// TIA Portal V15.1 export
// export: Created 2024-05-17T05:38:33.7575808Z, ExportSetting WithDefaults, DisplayName Totally Integrated Automation Portal, DisplayVersion V15.1 Update 5, DisplayName TIA Portal Openness, DisplayVersion V15.1 Update 5, DisplayName SINAMICS Startdrive Advanced, DisplayVersion V15.1, DisplayName G130, G150, S120, S150, SINAMICS MV, S210, DisplayVersion V15.1, DisplayName G110M, G120, G120C, G120D, G120P, DisplayVersion V15.1, DisplayName STEP 7 Professional, DisplayVersion V15.1 Update 5, DisplayName STEP 7 Safety, DisplayVersion V15.1, DisplayName WinCC Professional, DisplayVersion V15.1 Update 5, DisplayName SIMATIC Visualization Architect, DisplayVersion V15.1
FUNCTION_BLOCK "LProcMonStabValv"   // FB1701, FBD
TITLE = LProcMonStabValv
{ S7_Optimized_Access := 'FALSE' }
AUTHOR : VCC
FAMILY : ProcEqp
NAME : ProcValv
VERSION : 1.0
// ================================================================================
// This module is used to activate a monostable valve. It includes its own Mode 
// function. There is the possibility to use it normally open or normally closed, 
// with or without closed and open detections.
// ================================================================================
// stored: AutoNumber false, IsIECCheckEnabled false, SetENOAutomatically False, UDAEnableTagReadback false
   VAR_INPUT
      I_MaxTime { ExternalAccessible := 'False'; ExternalVisible := 'False'; ExternalWritable := 'False'} : DInt;   // Maximum Time to get Set and reset detections
      I_DetSet { ExternalAccessible := 'False'; ExternalVisible := 'False'; ExternalWritable := 'False'} : Bool;   // Detection SET
      I_DetReset { ExternalAccessible := 'False'; ExternalVisible := 'False'; ExternalWritable := 'False'} : Bool;   // Detection RESET
      I_EnableAlarm { ExternalAccessible := 'False'; ExternalVisible := 'False'; ExternalWritable := 'False'} : Bool;   // Enable Alarm for the Acof detections
      I_AutoReq { ExternalAccessible := 'False'; ExternalVisible := 'False'; ExternalWritable := 'False'} : Bool;   // Auto Request from equation or Sequence
      I_InterlockOk { ExternalAccessible := 'False'; ExternalVisible := 'False'; ExternalWritable := 'False'} : Bool;   // Interlock
      I_PBSetPBResetAllAutoSel { ExternalAccessible := 'False'; ExternalVisible := 'False'; ExternalWritable := 'False'} : Struct   // Set PB activated - Reset PB activated - All HMI Auto selected
         HMI1SetPB { ExternalAccessible := 'False'; ExternalVisible := 'False'; ExternalWritable := 'False'} : Bool;   // Set PB activated on HMI1
         HMI1ResetPB { ExternalAccessible := 'False'; ExternalVisible := 'False'; ExternalWritable := 'False'} : Bool;   // Reset PB activated on HMI1
         HMI1AllHMIAutoSel { ExternalAccessible := 'False'; ExternalVisible := 'False'; ExternalWritable := 'False'} : Bool;   // All HMI Auto selected on HMI1
         HMI2SetPB { ExternalAccessible := 'False'; ExternalVisible := 'False'; ExternalWritable := 'False'} : Bool;   // Set PB activated on HMI2
         HMI2ResetPB { ExternalAccessible := 'False'; ExternalVisible := 'False'; ExternalWritable := 'False'} : Bool;   // Reset PB activated on HMI2
         HMI2AllHMIAutoSel { ExternalAccessible := 'False'; ExternalVisible := 'False'; ExternalWritable := 'False'} : Bool;   // All HMI Auto selected on HMI2
         HMI3SetPB { ExternalAccessible := 'False'; ExternalVisible := 'False'; ExternalWritable := 'False'} : Bool;   // Set PB activated on HMI3
         HMI3ResetPB { ExternalAccessible := 'False'; ExternalVisible := 'False'; ExternalWritable := 'False'} : Bool;   // Reset PB activated on HMI3
         HMI3AllHMIAutoSel { ExternalAccessible := 'False'; ExternalVisible := 'False'; ExternalWritable := 'False'} : Bool;   // All HMI Auto selected on HMI3
         HMI4SetPB { ExternalAccessible := 'False'; ExternalVisible := 'False'; ExternalWritable := 'False'} : Bool;   // Set PB activated on HMI4
         HMI4ResetPB { ExternalAccessible := 'False'; ExternalVisible := 'False'; ExternalWritable := 'False'} : Bool;   // Reset PB activated on HMI4
         HMI4AllHMIAutoSel { ExternalAccessible := 'False'; ExternalVisible := 'False'; ExternalWritable := 'False'} : Bool;   // All HMI Auto selected on HMI4
         HMI5SetPB { ExternalAccessible := 'False'; ExternalVisible := 'False'; ExternalWritable := 'False'} : Bool;   // Set PB activated on HMI5
         HMI5ResetPB { ExternalAccessible := 'False'; ExternalVisible := 'False'; ExternalWritable := 'False'} : Bool;   // Reset PB activated on HMI5
         HMI5AllHMIAutoSel { ExternalAccessible := 'False'; ExternalVisible := 'False'; ExternalWritable := 'False'} : Bool;   // All HMI Auto selected on HMI5
         StartPBSel { ExternalAccessible := 'False'; ExternalVisible := 'False'; ExternalWritable := 'False'} : Bool;   // Start is activated
         AlarmResetPBSel { ExternalAccessible := 'False'; ExternalVisible := 'False'; ExternalWritable := 'False'} : Bool;   // Alarm reset is activated
      END_STRUCT;
      I_UpperLevelAlarmA { ExternalAccessible := 'False'; ExternalVisible := 'False'; ExternalWritable := 'False'} : Bool;   // Alarm A active from the top level
      I_UpperLevelAlarmB { ExternalAccessible := 'False'; ExternalVisible := 'False'; ExternalWritable := 'False'} : Bool;   // Alarm B active from the top level
      C_EnableSetResetHMI { ExternalAccessible := 'False'; ExternalVisible := 'False'; ExternalWritable := 'False'} : Bool;   // Enable Set-Reset functions from HMI
      C_ManualForcedUsed { ExternalAccessible := 'False'; ExternalVisible := 'False'; ExternalWritable := 'False'} : Bool;   // Manual Forced is used (=true)
      C_SelfHolding { ExternalAccessible := 'False'; ExternalVisible := 'False'; ExternalWritable := 'False'} : Bool := TRUE;   // Enable SelfHolding Command
      C_DetSetUsed { ExternalAccessible := 'False'; ExternalVisible := 'False'; ExternalWritable := 'False'} : Bool;   // Detection SET used (true=used)
      C_DetResetUsed { ExternalAccessible := 'False'; ExternalVisible := 'False'; ExternalWritable := 'False'} : Bool;   // Detection RESET used (true=used)
      C_ValveNO { ExternalAccessible := 'False'; ExternalVisible := 'False'; ExternalWritable := 'False'} : Bool;   // Valve Normally Open (NO=true)
   END_VAR
   VAR_OUTPUT
      O_ValveCmd { ExternalAccessible := 'False'; ExternalVisible := 'False'; ExternalWritable := 'False'} : Bool;   // Valve Command
      O_AlarmABCondition { ExternalAccessible := 'False'; ExternalVisible := 'False'; ExternalWritable := 'False'} : Bool;   // Alarm AB condition
      O_AlarmA { ExternalAccessible := 'False'; ExternalVisible := 'False'; ExternalWritable := 'False'} : Bool;   // Summary Alarm A from the Valve
      O_AlarmB { ExternalAccessible := 'False'; ExternalVisible := 'False'; ExternalWritable := 'False'} : Bool;   // Summary Alarm B from the Valve
      O_AlarmC { ExternalAccessible := 'False'; ExternalVisible := 'False'; ExternalWritable := 'False'} : Bool;   // Summary Alarm C from the Valve
      O_AlarmD { ExternalAccessible := 'False'; ExternalVisible := 'False'; ExternalWritable := 'False'} : Bool;   // Summary Alarm D from the Valve
      H_IAnim { ExternalAccessible := 'False'; ExternalVisible := 'False'; ExternalWritable := 'False'} : Word;   // HMI Animation of the icon
      H_AlarmWord { ExternalAccessible := 'False'; ExternalVisible := 'False'; ExternalWritable := 'False'} : DWord;   // Alarm Word
   END_VAR
   VAR DB_SPECIFIC
      AB_OverTimeAutoSel { ExternalAccessible := 'False'; ExternalVisible := 'False'; ExternalWritable := 'False'} : Bool;   // Alarm Overtime Auto selected
      AB_AcofDetSet { ExternalAccessible := 'False'; ExternalVisible := 'False'; ExternalWritable := 'False'} : Bool;   // Acof Fault Set detection
      AB_AcofDetReset { ExternalAccessible := 'False'; ExternalVisible := 'False'; ExternalWritable := 'False'} : Bool;   // Acof Fault Reset detection
      AD_InterlockAlarm { ExternalAccessible := 'False'; ExternalVisible := 'False'; ExternalWritable := 'False'} : Bool;   // Interlock Fault
      H_HMIModeCmd : Word;   // Mode commands from HMI
      H_ActiveHMI : Int;   // Active HMI
      H_NameActiveHMI : String[25];   // Name of the Active HMI
      H_Out : Struct   // HMI
         DetSetIAnim : Word;   // HMI Animation of the Detection
         DetResetIAnim : Word;   // HMI Animation of the Detection
         OutputIAnim : Word;   // HMI Animation of the output
         Anim : Word;   // HMI Animation of the object
         Anim2 : Word;   // HMI Animation of the object
         Anim3 : Bool;   // HMI Animation bool
         DBnr : Int;   // HMI Animation DB number
      END_STRUCT;
      OverTimeAutoSelCond { ExternalAccessible := 'False'; ExternalVisible := 'False'; ExternalWritable := 'False'} : Bool;   // Overtime Auto selected condition
      AcofDetSetCond { ExternalAccessible := 'False'; ExternalVisible := 'False'; ExternalWritable := 'False'} : Bool;   // Acof Detection set condition
      AcofDetResetCond { ExternalAccessible := 'False'; ExternalVisible := 'False'; ExternalWritable := 'False'} : Bool;   // Acof Detection reset condition
      AutoMode { ExternalAccessible := 'False'; ExternalVisible := 'False'; ExternalWritable := 'False'} : Bool;   // Auto mode
      ManualMode { ExternalAccessible := 'False'; ExternalVisible := 'False'; ExternalWritable := 'False'} : Bool;   // Manual mode
      AutoModeSel { ExternalAccessible := 'False'; ExternalVisible := 'False'; ExternalWritable := 'False'} : Bool;   // Auto Mode Selection from HMI
      ManualModeSel { ExternalAccessible := 'False'; ExternalVisible := 'False'; ExternalWritable := 'False'} : Bool;   // Manual Mode Selection from HMI
      ForcedMan { ExternalAccessible := 'False'; ExternalVisible := 'False'; ExternalWritable := 'False'} : Bool;   // Forced manual active
      ForcedManTimer { ExternalAccessible := 'False'; ExternalVisible := 'False'; ExternalWritable := 'False'} : Bool;   // Forced manual timer
      HMISetCmd { ExternalAccessible := 'False'; ExternalVisible := 'False'; ExternalWritable := 'False'} : Bool;   // Set Command on HMI
      HMIResetCmd { ExternalAccessible := 'False'; ExternalVisible := 'False'; ExternalWritable := 'False'} : Bool;   // Reset Command on HMI
      H_FncSelInHMI { ExternalAccessible := 'False'; ExternalVisible := 'False'; ExternalWritable := 'False'} : Bool;   // Manual selection from HMI
      SetPBMan { ExternalAccessible := 'False'; ExternalVisible := 'False'; ExternalWritable := 'False'} : Bool;   // Set pushbutton is activated in manual
      ResetPBMan { ExternalAccessible := 'False'; ExternalVisible := 'False'; ExternalWritable := 'False'} : Bool;   // Reset pushbutton is activated in manual
      AllHMIAutoSel { ExternalAccessible := 'False'; ExternalVisible := 'False'; ExternalWritable := 'False'} : Bool;   // All HMI Auto selected
      CmdRequest { ExternalAccessible := 'False'; ExternalVisible := 'False'; ExternalWritable := 'False'} : Bool;   // Command request to activate the component
      OvTimeAutoSel { ExternalAccessible := 'False'; ExternalVisible := 'False'; ExternalWritable := 'False'} : Bool;   // Alarm Overtime Auto selected and Component activated
      AlarmA { ExternalAccessible := 'False'; ExternalVisible := 'False'; ExternalWritable := 'False'} : Bool;   // Summation Alarm A of roller.
      AlarmB { ExternalAccessible := 'False'; ExternalVisible := 'False'; ExternalWritable := 'False'} : Bool;   // Summation Alarm B of roller.
      AlarmC { ExternalAccessible := 'False'; ExternalVisible := 'False'; ExternalWritable := 'False'} : Bool;   // Summation Alarm C of roller.
      AlarmD { ExternalAccessible := 'False'; ExternalVisible := 'False'; ExternalWritable := 'False'} : Bool;   // Summation Alarm D of roller.
      DBnr { ExternalAccessible := 'False'; ExternalVisible := 'False'; ExternalWritable := 'False'} : Int;   // HMI DB number
   END_VAR
   VAR
      DetSet { ExternalAccessible := 'False'; ExternalVisible := 'False'; ExternalWritable := 'False'; S7_SetPoint := 'True'} : "LProcAcofDet";   // Acof Detection Set
      DetReset { ExternalAccessible := 'False'; ExternalVisible := 'False'; ExternalWritable := 'False'; S7_SetPoint := 'True'} : "LProcAcofDet";   // Acof Detection Reset
      Modes { ExternalAccessible := 'False'; ExternalVisible := 'False'; ExternalWritable := 'False'; S7_SetPoint := 'True'} : "LProcObjectMode";
   END_VAR
   VAR DB_SPECIFIC
      CheckActiveHMI { ExternalAccessible := 'False'; ExternalVisible := 'False'; ExternalWritable := 'False'; S7_SetPoint := 'True'} : TP_TIME;   // Timer
      CheckActiveHMI_1 { ExternalAccessible := 'False'; ExternalVisible := 'False'; ExternalWritable := 'False'; S7_SetPoint := 'True'} : TP_TIME;   // Timer
      CheckActiveHMI_2 { ExternalAccessible := 'False'; ExternalVisible := 'False'; ExternalWritable := 'False'; S7_SetPoint := 'True'} : TON_TIME;   // Timer
      CheckActiveHMI_3 { ExternalAccessible := 'False'; ExternalVisible := 'False'; ExternalWritable := 'False'; S7_SetPoint := 'True'} : TON_TIME;   // Timer
   END_VAR
BEGIN

NETWORK
TITLE = **** 1 - Inputs **** DB number
// DB number
      L     DINO;
      T     #DBnr;

REGION Network 2: **** 2.2 - Alarms - Alarm Generation **** Interlock Alarm
   // Interlock Alarm
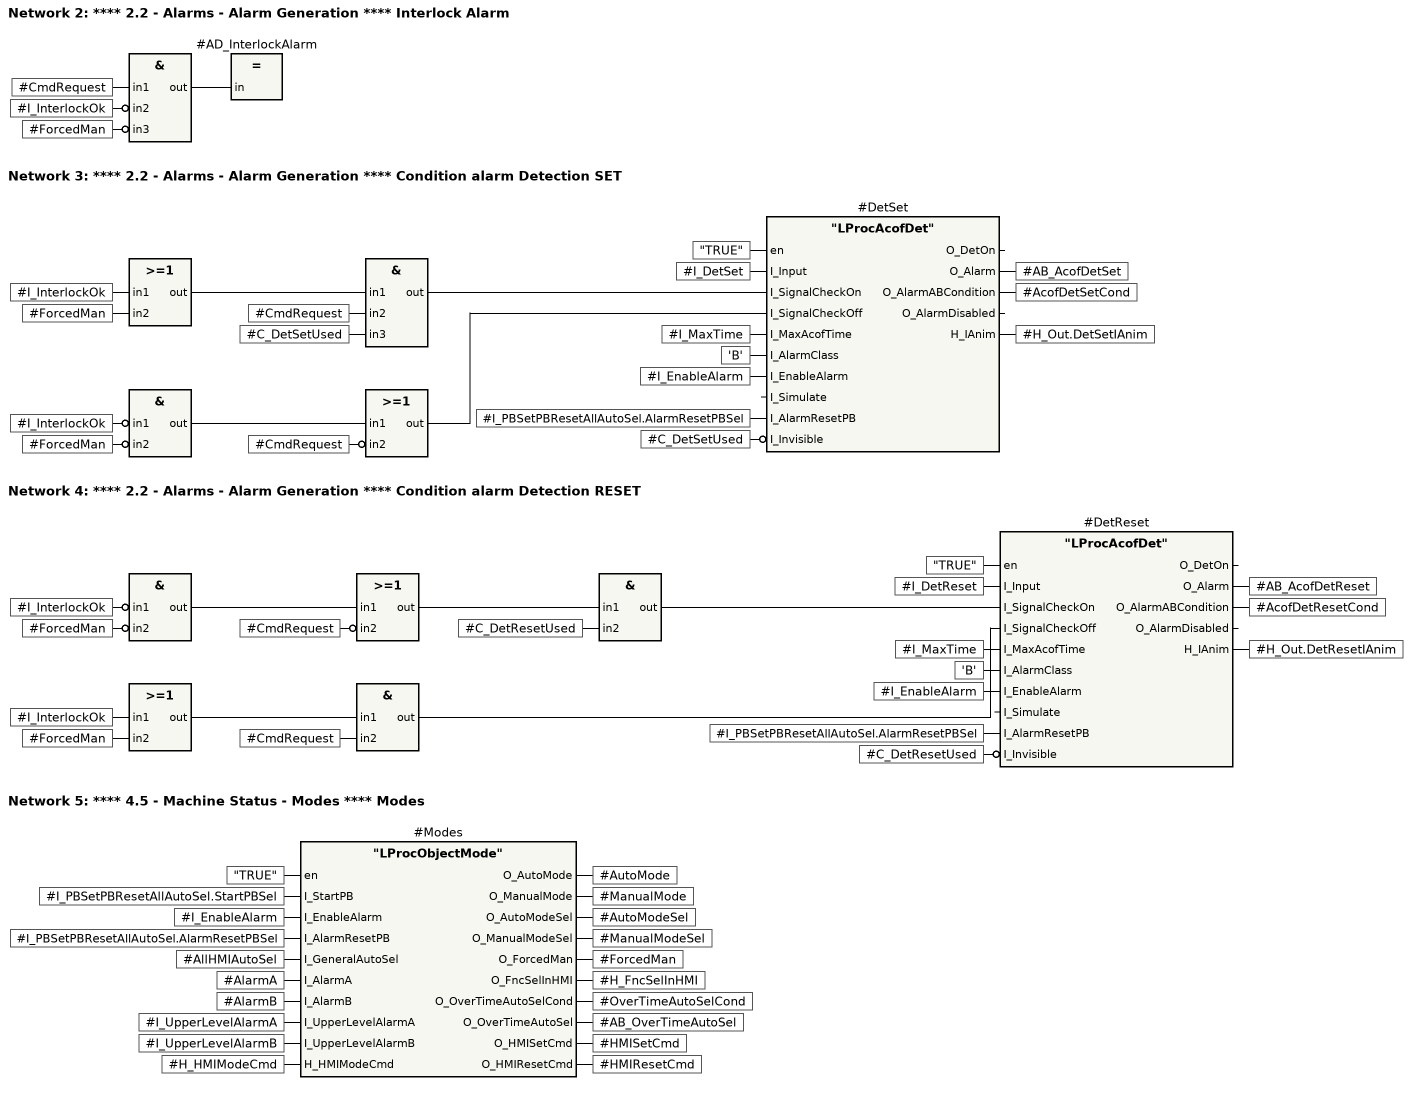
   #AD_InterlockAlarm := #CmdRequest AND NOT #I_InterlockOk AND NOT #ForcedMan;
END_REGION

REGION Network 3: **** 2.2 - Alarms - Alarm Generation **** Condition alarm Detection SET
   // Condition alarm Detection SET
   IF "TRUE" THEN
       #DetSet(I_Input := #I_DetSet,   // "LProcAcofDet"
               I_SignalCheckOn := (#I_InterlockOk OR #ForcedMan) AND #CmdRequest AND #C_DetSetUsed,
               I_SignalCheckOff := (NOT #I_InterlockOk AND NOT #ForcedMan) OR NOT #CmdRequest,
               I_MaxAcofTime := #I_MaxTime,
               I_AlarmClass := 'B',
               I_EnableAlarm := #I_EnableAlarm,
               I_AlarmResetPB := #I_PBSetPBResetAllAutoSel.AlarmResetPBSel,
               I_Invisible := NOT #C_DetSetUsed,
               O_Alarm => #AB_AcofDetSet,
               O_AlarmABCondition => #AcofDetSetCond,
               H_IAnim => #H_Out.DetSetIAnim);
   END_IF;
END_REGION

REGION Network 4: **** 2.2 - Alarms - Alarm Generation **** Condition alarm Detection RESET
   // Condition alarm Detection RESET
   IF "TRUE" THEN
       #DetReset(I_Input := #I_DetReset,   // "LProcAcofDet"
                 I_SignalCheckOn := ((NOT #I_InterlockOk AND NOT #ForcedMan) OR NOT #CmdRequest) AND #C_DetResetUsed,
                 I_SignalCheckOff := (#I_InterlockOk OR #ForcedMan) AND #CmdRequest,
                 I_MaxAcofTime := #I_MaxTime,
                 I_AlarmClass := 'B',
                 I_EnableAlarm := #I_EnableAlarm,
                 I_AlarmResetPB := #I_PBSetPBResetAllAutoSel.AlarmResetPBSel,
                 I_Invisible := NOT #C_DetResetUsed,
                 O_Alarm => #AB_AcofDetReset,
                 O_AlarmABCondition => #AcofDetResetCond,
                 H_IAnim => #H_Out.DetResetIAnim);
   END_IF;
END_REGION

REGION Network 5: **** 4.5 - Machine Status - Modes **** Modes
   // Modes
   IF "TRUE" THEN
       #Modes(I_StartPB := #I_PBSetPBResetAllAutoSel.StartPBSel,   // "LProcObjectMode"
              I_EnableAlarm := #I_EnableAlarm,
              I_AlarmResetPB := #I_PBSetPBResetAllAutoSel.AlarmResetPBSel,
              I_GeneralAutoSel := #AllHMIAutoSel,
              I_AlarmA := #AlarmA,
              I_AlarmB := #AlarmB,
              I_UpperLevelAlarmA := #I_UpperLevelAlarmA,
              I_UpperLevelAlarmB := #I_UpperLevelAlarmB,
              H_HMIModeCmd := #H_HMIModeCmd,
              O_AutoMode => #AutoMode,
              O_ManualMode => #ManualMode,
              O_AutoModeSel => #AutoModeSel,
              O_ManualModeSel => #ManualModeSel,
              O_ForcedMan => #ForcedMan,
              O_FncSelInHMI => #H_FncSelInHMI,
              O_OverTimeAutoSelCond => #OverTimeAutoSelCond,
              O_OverTimeAutoSel => #AB_OverTimeAutoSel,
              O_HMISetCmd => #HMISetCmd,
              O_HMIResetCmd => #HMIResetCmd);
   END_IF;
END_REGION

REGION Network 6: **** 4.6 - Machine status - Indications **** Valve Animation for HMI
   // Valve Animation for HMI
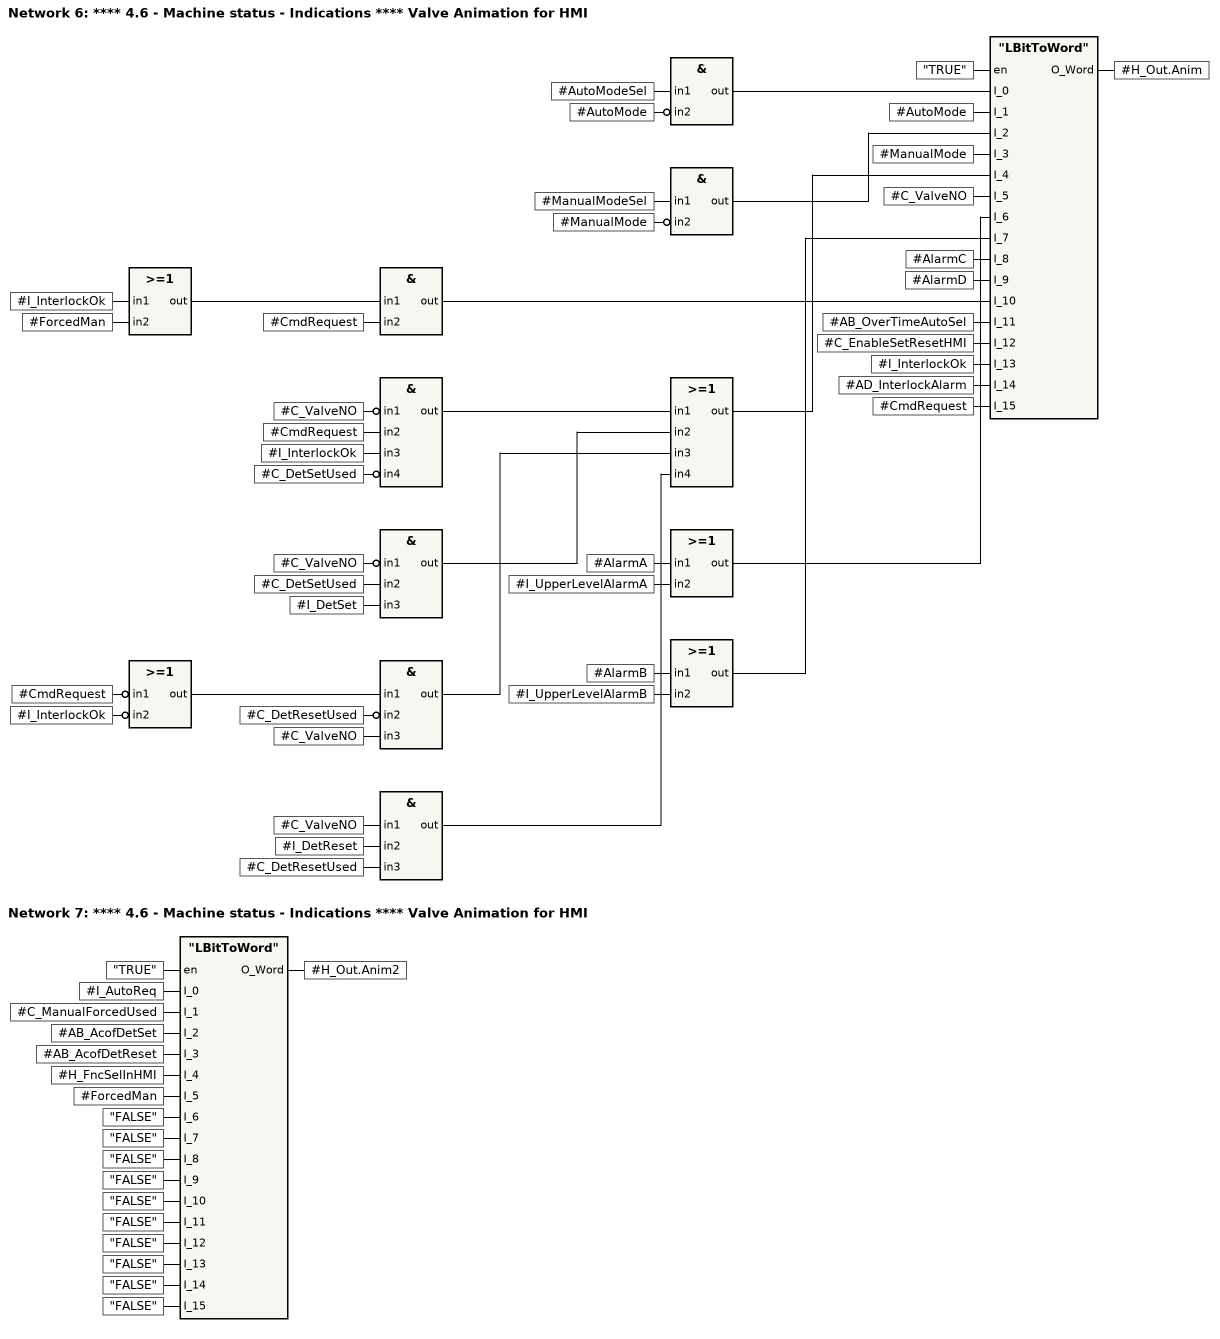
   IF "TRUE" THEN
       "LBitToWord"(I_0 := #AutoModeSel AND NOT #AutoMode,
                    I_1 := #AutoMode,
                    I_2 := #ManualModeSel AND NOT #ManualMode,
                    I_3 := #ManualMode,
                    I_4 := (NOT #C_ValveNO AND #CmdRequest AND #I_InterlockOk AND NOT #C_DetSetUsed) OR (NOT #C_ValveNO AND #C_DetSetUsed AND #I_DetSet) OR ((NOT #CmdRequest OR NOT #I_InterlockOk) AND NOT #C_DetResetUsed AND #C_ValveNO) OR (#C_ValveNO AND #I_DetReset AND #C_DetResetUsed),
                    I_5 := #C_ValveNO,
                    I_6 := #AlarmA OR #I_UpperLevelAlarmA,
                    I_7 := #AlarmB OR #I_UpperLevelAlarmB,
                    I_8 := #AlarmC,
                    I_9 := #AlarmD,
                    I_10 := (#I_InterlockOk OR #ForcedMan) AND #CmdRequest,
                    I_11 := #AB_OverTimeAutoSel,
                    I_12 := #C_EnableSetResetHMI,
                    I_13 := #I_InterlockOk,
                    I_14 := #AD_InterlockAlarm,
                    I_15 := #CmdRequest,
                    O_Word => #H_Out.Anim);
   END_IF;
END_REGION

REGION Network 7: **** 4.6 - Machine status - Indications **** Valve Animation for HMI
   // Valve Animation for HMI
   IF "TRUE" THEN
       "LBitToWord"(I_0 := #I_AutoReq,
                    I_1 := #C_ManualForcedUsed,
                    I_2 := #AB_AcofDetSet,
                    I_3 := #AB_AcofDetReset,
                    I_4 := #H_FncSelInHMI,
                    I_5 := #ForcedMan,
                    I_6 := "FALSE",
                    I_7 := "FALSE",
                    I_8 := "FALSE",
                    I_9 := "FALSE",
                    I_10 := "FALSE",
                    I_11 := "FALSE",
                    I_12 := "FALSE",
                    I_13 := "FALSE",
                    I_14 := "FALSE",
                    I_15 := "FALSE",
                    O_Word => #H_Out.Anim2);
   END_IF;
END_REGION

REGION Network 8: **** 4.6 - Machine status - Indications **** Valve Animation for HMI
   // Valve Animation for HMI
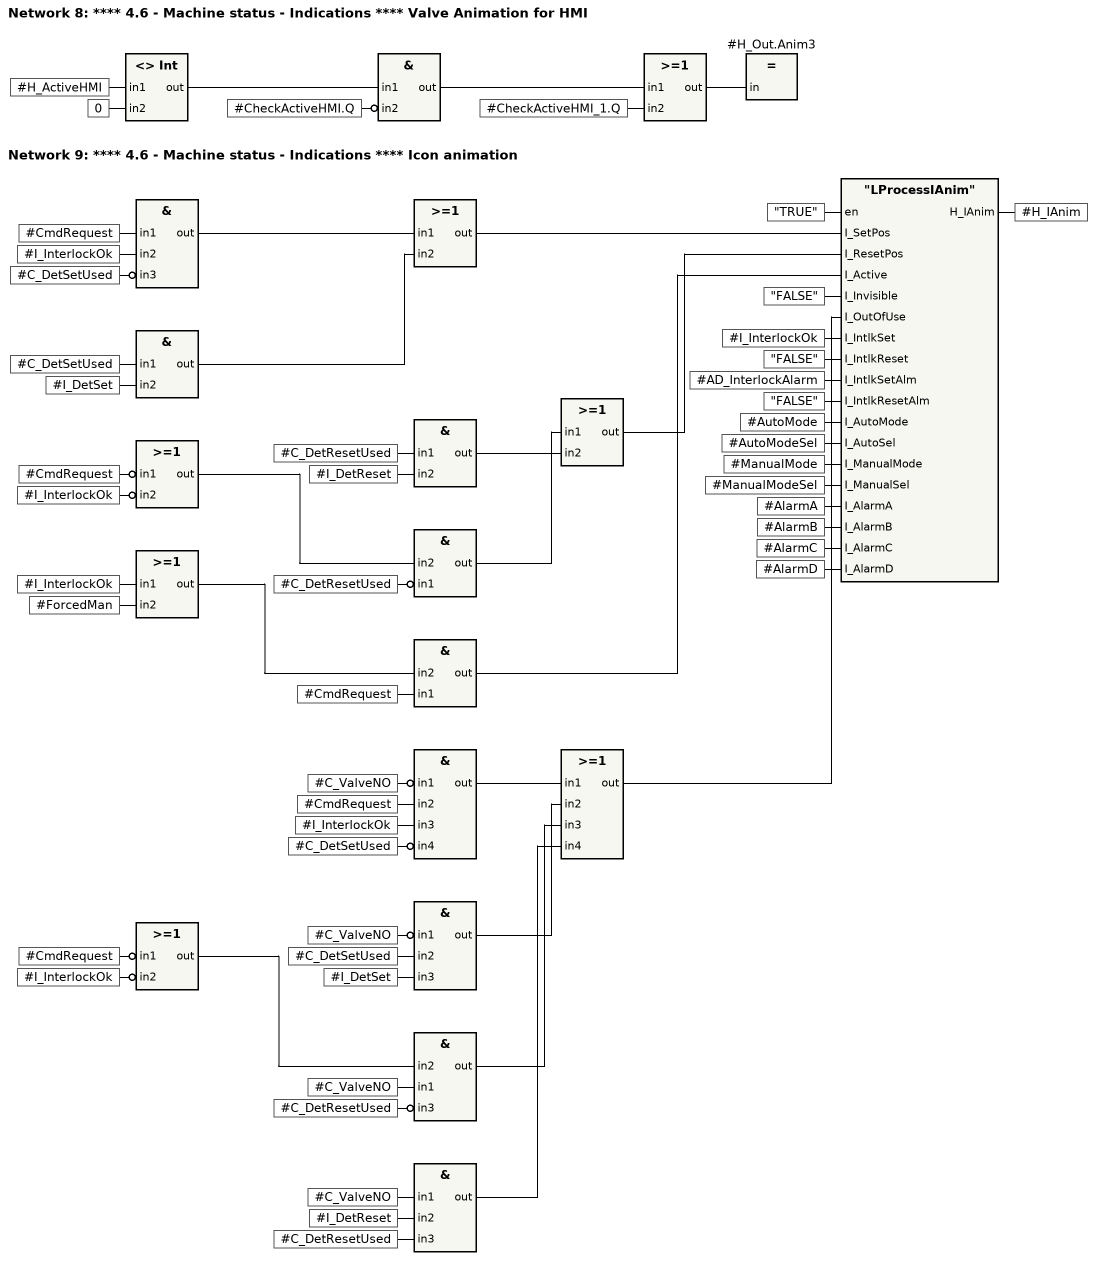
   #H_Out.Anim3 := ((#H_ActiveHMI <> 0) AND NOT #CheckActiveHMI.Q) OR #CheckActiveHMI_1.Q;
END_REGION

REGION Network 9: **** 4.6 - Machine status - Indications **** Icon animation
   // Icon animation
   IF "TRUE" THEN
       "LProcessIAnim"(I_SetPos := (#CmdRequest AND #I_InterlockOk AND NOT #C_DetSetUsed) OR (#C_DetSetUsed AND #I_DetSet),
                       I_ResetPos := ((NOT #CmdRequest OR NOT #I_InterlockOk) AND NOT #C_DetResetUsed) OR (#C_DetResetUsed AND #I_DetReset),
                       I_Active := (#I_InterlockOk OR #ForcedMan) AND #CmdRequest,
                       I_Invisible := "FALSE",
                       I_OutOfUse := (NOT #C_ValveNO AND #CmdRequest AND #I_InterlockOk AND NOT #C_DetSetUsed) OR (NOT #C_ValveNO AND #C_DetSetUsed AND #I_DetSet) OR ((NOT #CmdRequest OR NOT #I_InterlockOk) AND #C_ValveNO AND NOT #C_DetResetUsed) OR (#C_ValveNO AND #I_DetReset AND #C_DetResetUsed),
                       I_IntlkSet := #I_InterlockOk,
                       I_IntlkReset := "FALSE",
                       I_IntlkSetAlm := #AD_InterlockAlarm,
                       I_IntlkResetAlm := "FALSE",
                       I_AutoMode := #AutoMode,
                       I_AutoSel := #AutoModeSel,
                       I_ManualMode := #ManualMode,
                       I_ManualSel := #ManualModeSel,
                       I_AlarmA := #AlarmA,
                       I_AlarmB := #AlarmB,
                       I_AlarmC := #AlarmC,
                       I_AlarmD := #AlarmD,
                       H_IAnim => #H_IAnim);
   END_IF;
END_REGION

REGION Network 10: **** 4.6 - Machine status - Indications **** Valve Output animation
   // Valve Output animation
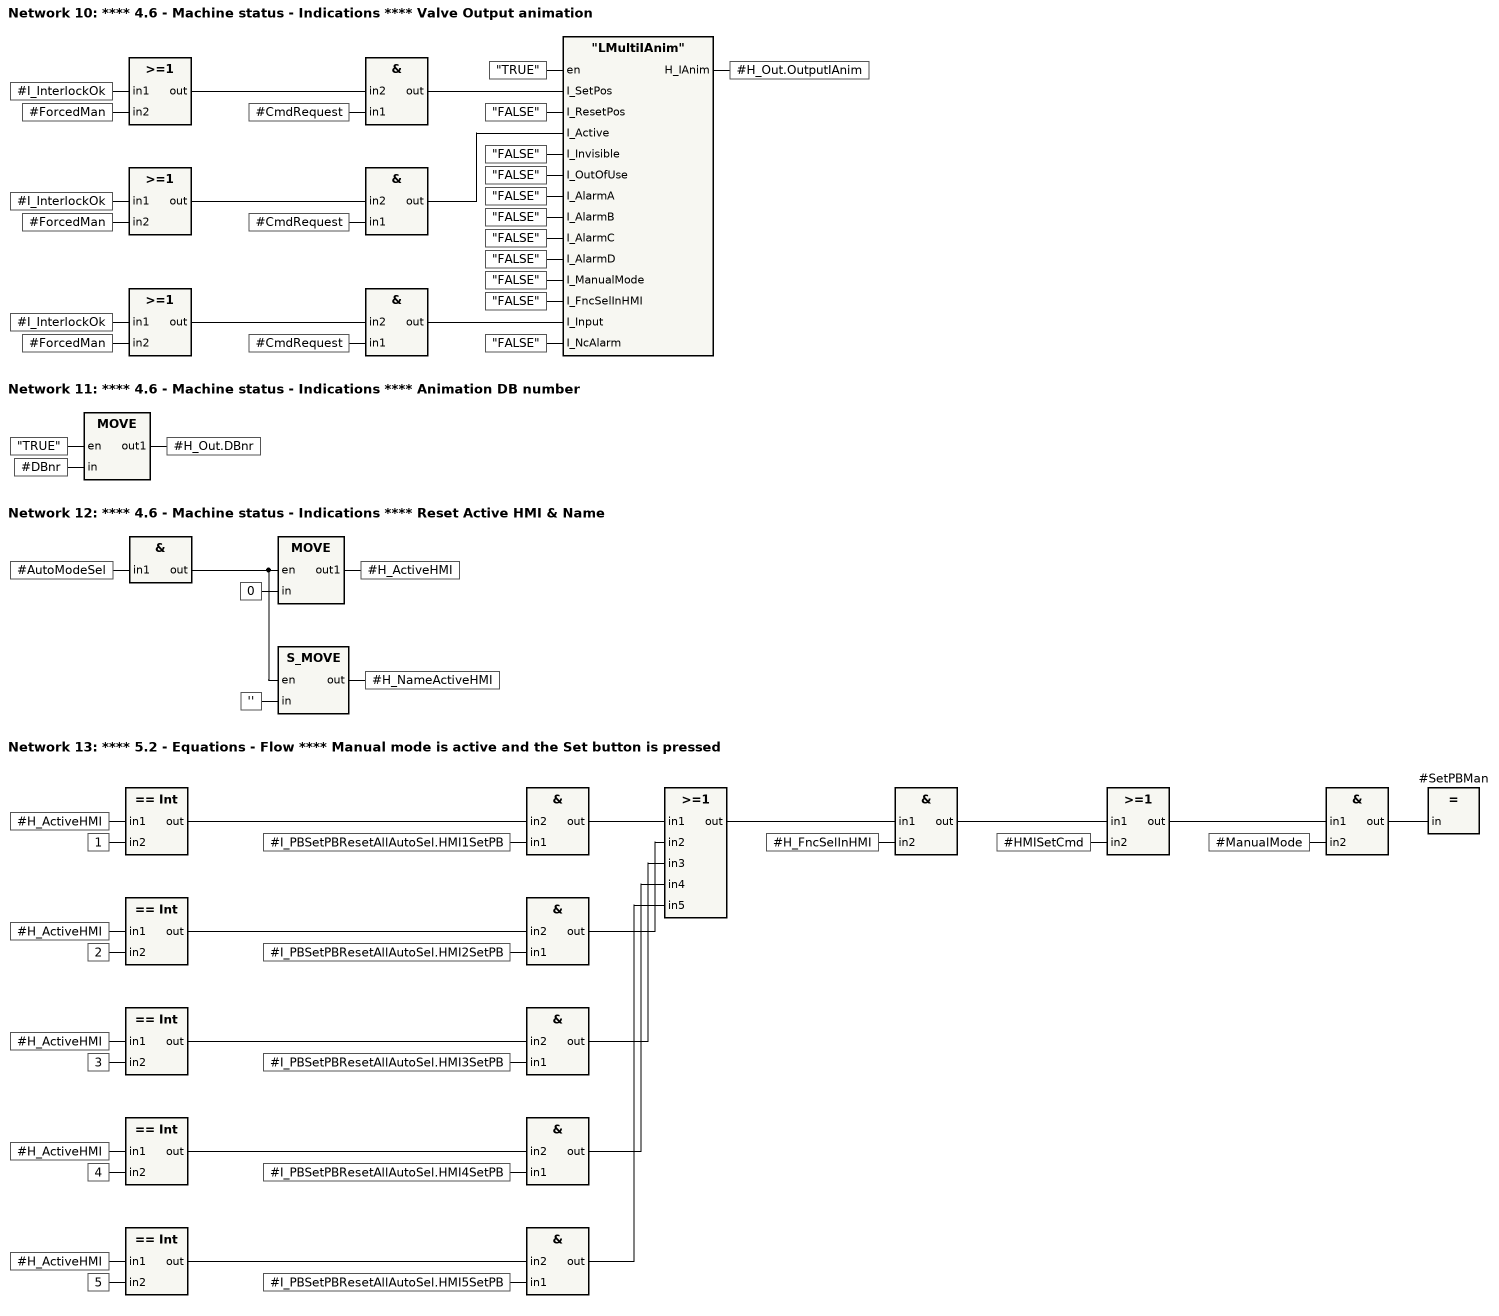
   IF "TRUE" THEN
       "LMultiIAnim"(I_SetPos := (#I_InterlockOk OR #ForcedMan) AND #CmdRequest,
                     I_ResetPos := "FALSE",
                     I_Active := (#I_InterlockOk OR #ForcedMan) AND #CmdRequest,
                     I_Invisible := "FALSE",
                     I_OutOfUse := "FALSE",
                     I_AlarmA := "FALSE",
                     I_AlarmB := "FALSE",
                     I_AlarmC := "FALSE",
                     I_AlarmD := "FALSE",
                     I_ManualMode := "FALSE",
                     I_FncSelInHMI := "FALSE",
                     I_Input := (#I_InterlockOk OR #ForcedMan) AND #CmdRequest,
                     I_NcAlarm := "FALSE",
                     H_IAnim => #H_Out.OutputIAnim);
   END_IF;
END_REGION

REGION Network 11: **** 4.6 - Machine status - Indications **** Animation DB number
   // Animation DB number
   IF "TRUE" THEN #H_Out.DBnr := #DBnr; END_IF;
END_REGION

REGION Network 12: **** 4.6 - Machine status - Indications **** Reset Active HMI & Name
   // Reset Active HMI & Name
   IF #AutoModeSel THEN
       #H_ActiveHMI := 0;
       #H_NameActiveHMI := '';
   END_IF;
END_REGION

REGION Network 13: **** 5.2 - Equations - Flow **** Manual mode is active and the Set button is pressed
   // Manual mode is active and the Set button is pressed
   #SetPBMan := (((((#H_ActiveHMI = 1) AND #I_PBSetPBResetAllAutoSel.HMI1SetPB) OR ((#H_ActiveHMI = 2) AND #I_PBSetPBResetAllAutoSel.HMI2SetPB) OR ((#H_ActiveHMI = 3) AND #I_PBSetPBResetAllAutoSel.HMI3SetPB) OR ((#H_ActiveHMI = 4) AND #I_PBSetPBResetAllAutoSel.HMI4SetPB) OR ((#H_ActiveHMI = 5) AND #I_PBSetPBResetAllAutoSel.HMI5SetPB)) AND #H_FncSelInHMI) OR #HMISetCmd) AND #ManualMode;
END_REGION

REGION Network 14: **** 5.2 - Equations - Flow **** Manual mode is active and the Reset button is pressed
   // Manual mode is active and the Reset button is pressed
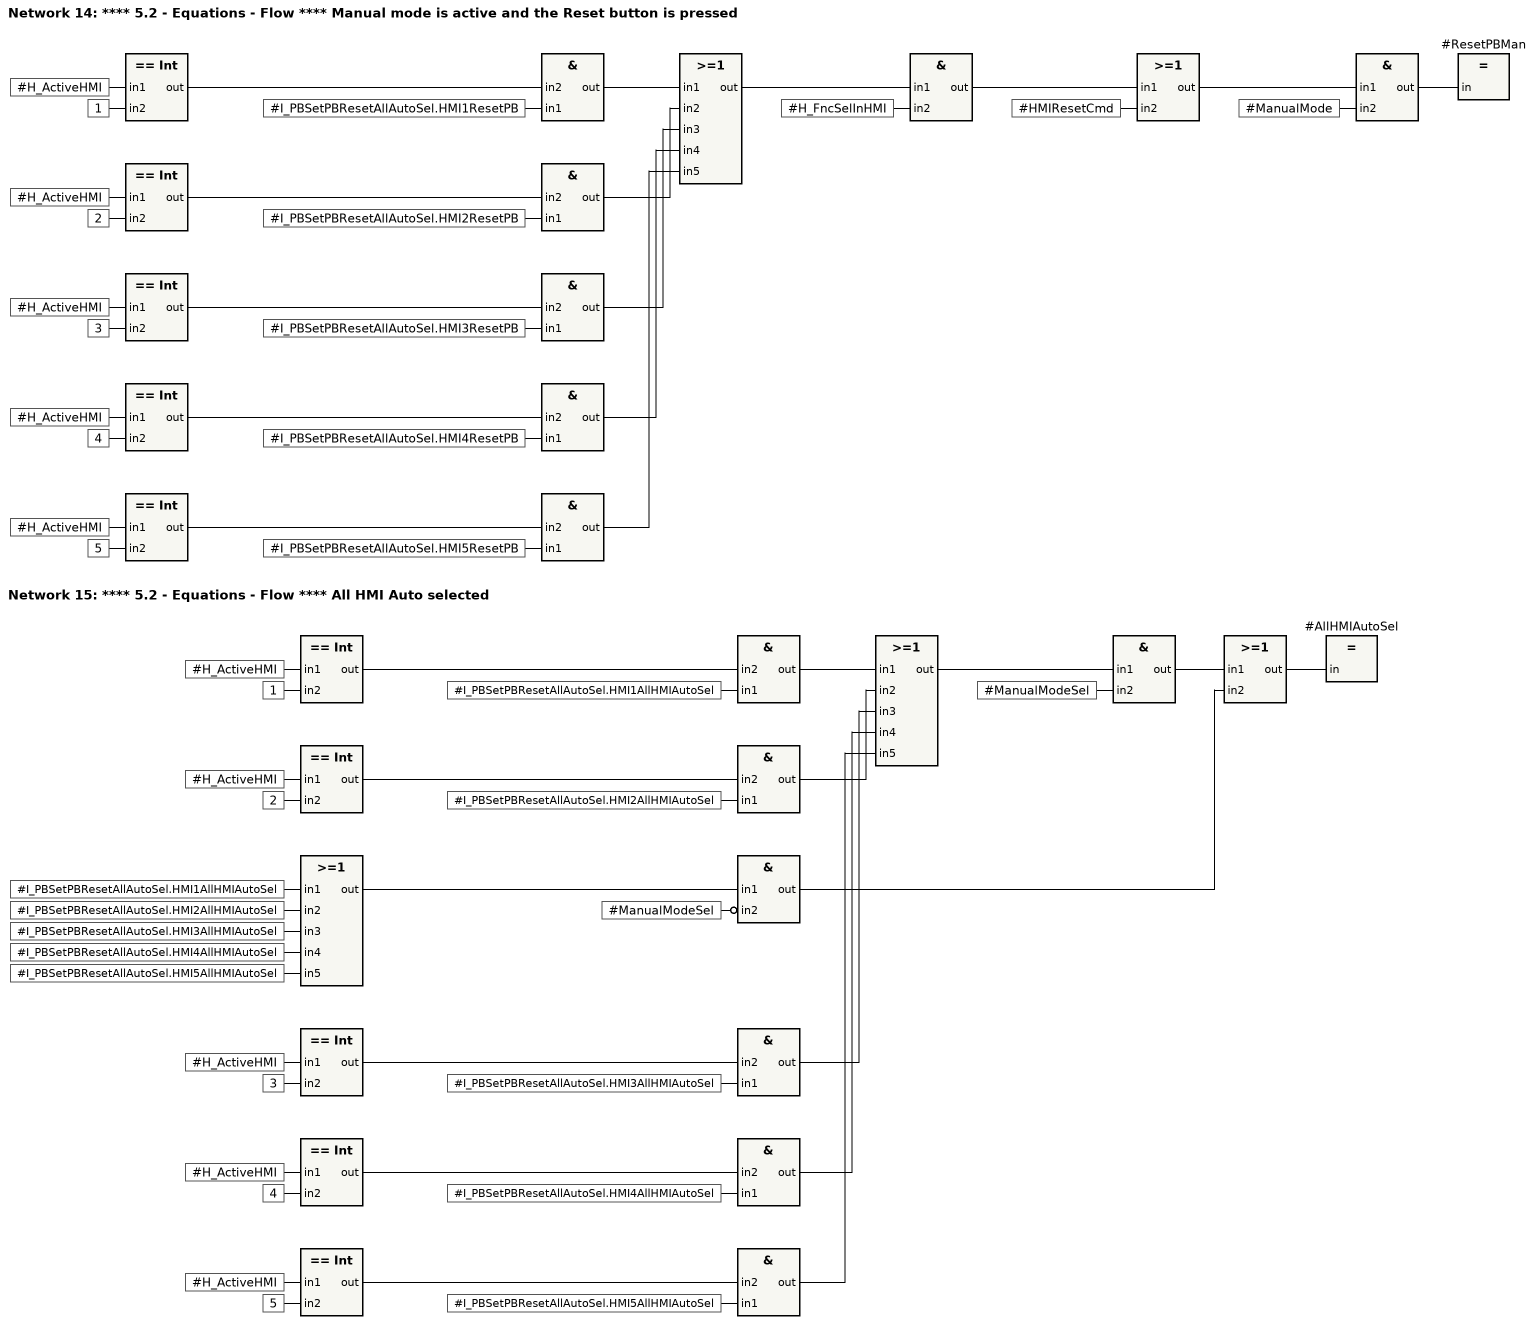
   #ResetPBMan := (((((#H_ActiveHMI = 1) AND #I_PBSetPBResetAllAutoSel.HMI1ResetPB) OR ((#H_ActiveHMI = 2) AND #I_PBSetPBResetAllAutoSel.HMI2ResetPB) OR ((#H_ActiveHMI = 3) AND #I_PBSetPBResetAllAutoSel.HMI3ResetPB) OR ((#H_ActiveHMI = 4) AND #I_PBSetPBResetAllAutoSel.HMI4ResetPB) OR ((#H_ActiveHMI = 5) AND #I_PBSetPBResetAllAutoSel.HMI5ResetPB)) AND #H_FncSelInHMI) OR #HMIResetCmd) AND #ManualMode;
END_REGION

REGION Network 15: **** 5.2 - Equations - Flow **** All HMI Auto selected
   // All HMI Auto selected
   #AllHMIAutoSel := ((((#H_ActiveHMI = 1) AND #I_PBSetPBResetAllAutoSel.HMI1AllHMIAutoSel) OR ((#H_ActiveHMI = 2) AND #I_PBSetPBResetAllAutoSel.HMI2AllHMIAutoSel) OR ((#H_ActiveHMI = 3) AND #I_PBSetPBResetAllAutoSel.HMI3AllHMIAutoSel) OR ((#H_ActiveHMI = 4) AND #I_PBSetPBResetAllAutoSel.HMI4AllHMIAutoSel) OR ((#H_ActiveHMI = 5) AND #I_PBSetPBResetAllAutoSel.HMI5AllHMIAutoSel)) AND #ManualModeSel) OR ((#I_PBSetPBResetAllAutoSel.HMI1AllHMIAutoSel OR #I_PBSetPBResetAllAutoSel.HMI2AllHMIAutoSel OR #I_PBSetPBResetAllAutoSel.HMI3AllHMIAutoSel OR #I_PBSetPBResetAllAutoSel.HMI4AllHMIAutoSel OR #I_PBSetPBResetAllAutoSel.HMI5AllHMIAutoSel) AND NOT #ManualModeSel);
END_REGION

REGION Network 16: **** 5.2 - Equations - Flow **** Check Active HMI again - HMI <> 0
   // Check Active HMI again
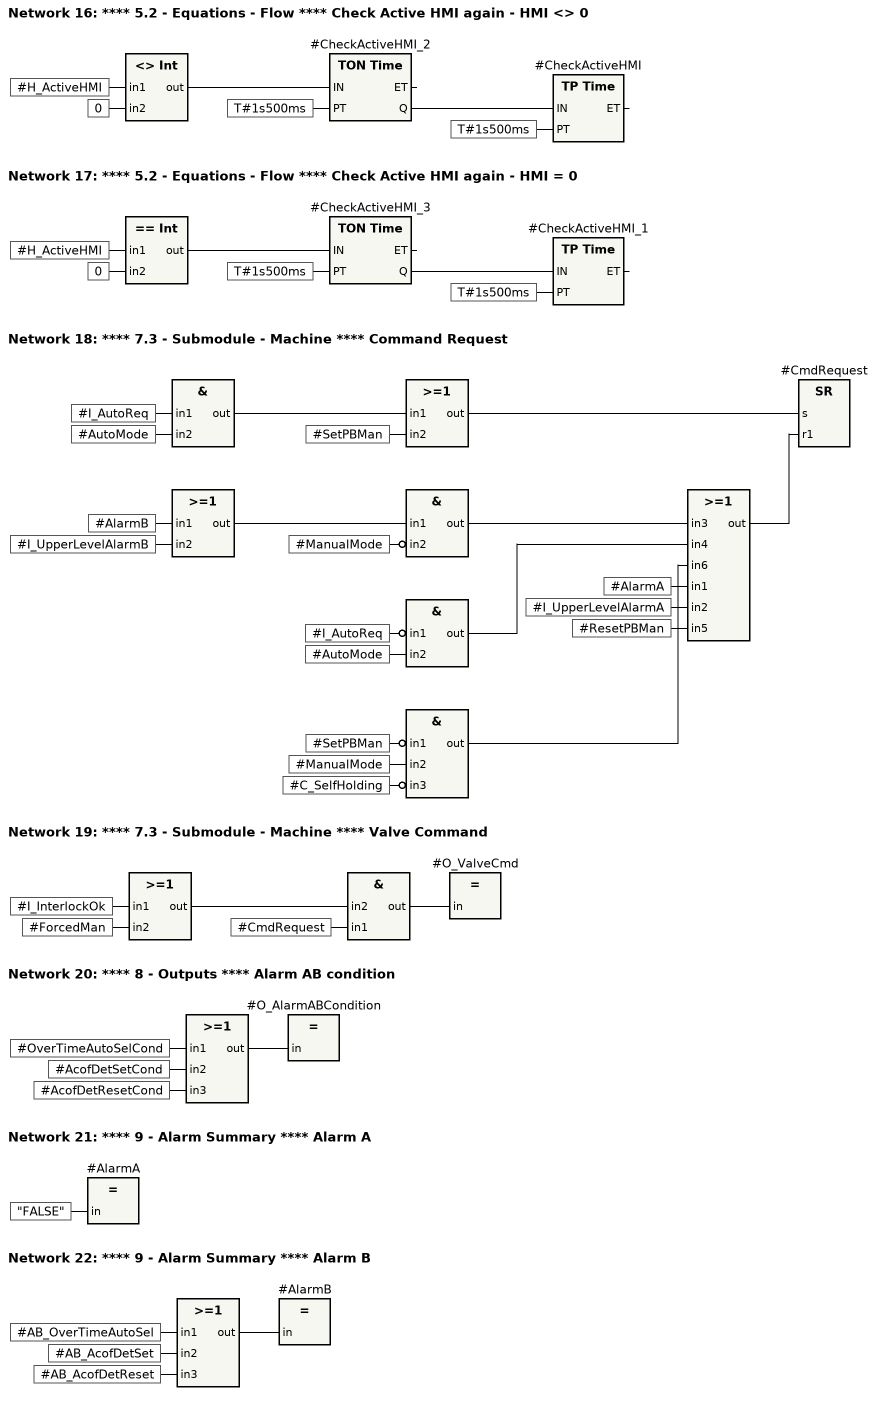
   #CheckActiveHMI_2(IN := #H_ActiveHMI <> 0, PT := T#1s500ms);   // TON
   #CheckActiveHMI(IN := #CheckActiveHMI_2.Q, PT := T#1s500ms);   // TP
END_REGION

REGION Network 17: **** 5.2 - Equations - Flow **** Check Active HMI again - HMI = 0
   // Check Active HMI again
   #CheckActiveHMI_3(IN := #H_ActiveHMI = 0, PT := T#1s500ms);   // TON
   #CheckActiveHMI_1(IN := #CheckActiveHMI_3.Q, PT := T#1s500ms);   // TP
END_REGION

REGION Network 18: **** 7.3 - Submodule - Machine **** Command Request
   // Command Request
   IF (#I_AutoReq AND #AutoMode) OR #SetPBMan THEN
       #CmdRequest := TRUE;   // SR flip-flop
   END_IF;
   IF ((#AlarmB OR #I_UpperLevelAlarmB) AND NOT #ManualMode) OR (NOT #I_AutoReq AND #AutoMode) OR (NOT #SetPBMan AND #ManualMode AND NOT #C_SelfHolding) OR #AlarmA OR #I_UpperLevelAlarmA OR #ResetPBMan THEN
       #CmdRequest := FALSE;
   END_IF;
END_REGION

REGION Network 19: **** 7.3 - Submodule - Machine **** Valve Command
   // Valve Command
   #O_ValveCmd := (#I_InterlockOk OR #ForcedMan) AND #CmdRequest;
END_REGION

REGION Network 20: **** 8 - Outputs **** Alarm AB condition
   // Alarm AB condition
   #O_AlarmABCondition := #OverTimeAutoSelCond OR #AcofDetSetCond OR #AcofDetResetCond;
END_REGION

REGION Network 21: **** 9 - Alarm Summary **** Alarm A
   // Summary of alarms A
   #AlarmA := "FALSE";
END_REGION

REGION Network 22: **** 9 - Alarm Summary **** Alarm B
   // Summary of alarms B
   #AlarmB := #AB_OverTimeAutoSel OR #AB_AcofDetSet OR #AB_AcofDetReset;
END_REGION

REGION Network 23: **** 9 - Alarm Summary **** Alarm C
   // Summary of alarms C
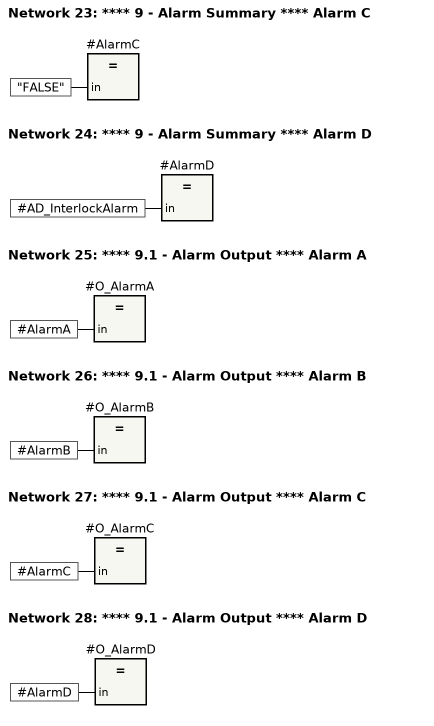
   #AlarmC := "FALSE";
END_REGION

REGION Network 24: **** 9 - Alarm Summary **** Alarm D
   // Summary of alarms D
   #AlarmD := #AD_InterlockAlarm;
END_REGION

REGION Network 25: **** 9.1 - Alarm Output **** Alarm A
   // Summary of alarms A
   #O_AlarmA := #AlarmA;
END_REGION

REGION Network 26: **** 9.1 - Alarm Output **** Alarm B
   // Summary of alarms B
   #O_AlarmB := #AlarmB;
END_REGION

REGION Network 27: **** 9.1 - Alarm Output **** Alarm C
   // Summary of alarms C
   #O_AlarmC := #AlarmC;
END_REGION

REGION Network 28: **** 9.1 - Alarm Output **** Alarm D
   // Summary of alarms D
   #O_AlarmD := #AlarmD;
END_REGION

REGION Network 29: **** 9.2 - Alarm DWord**** Alarm To DWord
   // Alarm Word
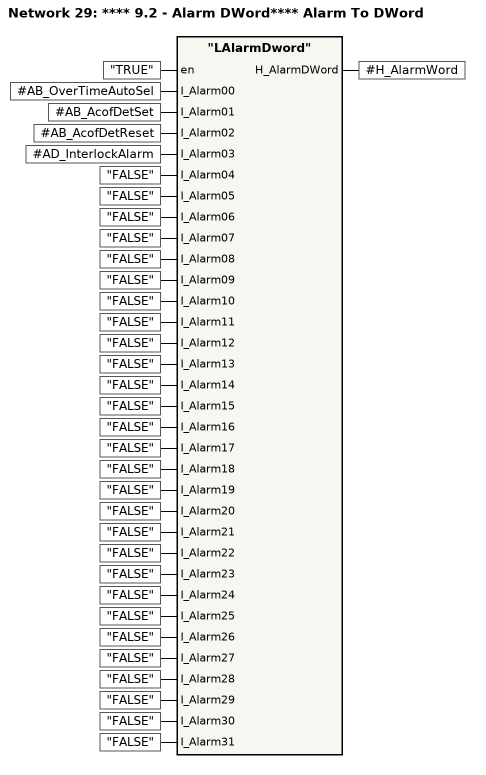
   IF "TRUE" THEN
       "LAlarmDword"(I_Alarm00 := #AB_OverTimeAutoSel,
                     I_Alarm01 := #AB_AcofDetSet,
                     I_Alarm02 := #AB_AcofDetReset,
                     I_Alarm03 := #AD_InterlockAlarm,
                     I_Alarm04 := "FALSE",
                     I_Alarm05 := "FALSE",
                     I_Alarm06 := "FALSE",
                     I_Alarm07 := "FALSE",
                     I_Alarm08 := "FALSE",
                     I_Alarm09 := "FALSE",
                     I_Alarm10 := "FALSE",
                     I_Alarm11 := "FALSE",
                     I_Alarm12 := "FALSE",
                     I_Alarm13 := "FALSE",
                     I_Alarm14 := "FALSE",
                     I_Alarm15 := "FALSE",
                     I_Alarm16 := "FALSE",
                     I_Alarm17 := "FALSE",
                     I_Alarm18 := "FALSE",
                     I_Alarm19 := "FALSE",
                     I_Alarm20 := "FALSE",
                     I_Alarm21 := "FALSE",
                     I_Alarm22 := "FALSE",
                     I_Alarm23 := "FALSE",
                     I_Alarm24 := "FALSE",
                     I_Alarm25 := "FALSE",
                     I_Alarm26 := "FALSE",
                     I_Alarm27 := "FALSE",
                     I_Alarm28 := "FALSE",
                     I_Alarm29 := "FALSE",
                     I_Alarm30 := "FALSE",
                     I_Alarm31 := "FALSE",
                     H_AlarmDWord => #H_AlarmWord);
   END_IF;
END_REGION
END_FUNCTION_BLOCK
